{attribute 'GeneratedUsingTerminal: EP6002-0002-0023'}
{attribute addProperty BoxType "EP6002-0002-0023"}
{attribute addProperty Description "EP6002-0002 Interface (RS232/422/485)"}
{attribute addProperty Physics "YY"}
{attribute addProperty Id "COM_TxPDO_Map_Inputs_Channel_1AT %I*COM_TxPDO_Map_Inputs_Channel_6C2FC20224COM_TxPDO_Map_Inputs_Channel_2AT %I*COM_TxPDO_Map_Inputs_Channel_6C2FC20224COM_RxPDO_Map_Outputs_Channel_1AT %Q*COM_RxPDO_Map_Outputs_Channel_5D00B5E724COM_RxPDO_Map_Outputs_Channel_2AT %Q*COM_RxPDO_Map_Outputs_Channel_5D00B5E724WcStateAT %I*WcState_9091E0EB2InfoDataAT %I*InfoData_32EB74EA10"}
{attribute addProperty CRC "2078717463"}
{attribute addProperty Size "108"}
TYPE EP6002_7BE6B617 EXTENDS EtcSlaveBoxBase_77A0E4A7 :
STRUCT
	{attribute addProperty Name "COM_TxPDO_Map_Inputs_Channel_1"}
	COM_TxPDO_Map_Inputs_Channel_1 : COM_TxPDO_Map_Inputs_Channel_6C2FC202;
	{attribute addProperty Name "COM_TxPDO_Map_Inputs_Channel_2"}
	COM_TxPDO_Map_Inputs_Channel_2 : COM_TxPDO_Map_Inputs_Channel_6C2FC202;
	{attribute addProperty Name "COM_RxPDO_Map_Outputs_Channel_1"}
	COM_RxPDO_Map_Outputs_Channel_1 : COM_RxPDO_Map_Outputs_Channel_5D00B5E7;
	{attribute addProperty Name "COM_RxPDO_Map_Outputs_Channel_2"}
	COM_RxPDO_Map_Outputs_Channel_2 : COM_RxPDO_Map_Outputs_Channel_5D00B5E7;
	{attribute addProperty Name "WcState"}
	WcState : WcState_9091E0EB;
	{attribute addProperty Name "InfoData"}
	InfoData : InfoData_32EB74EA;
END_STRUCT
END_TYPE

(* stored: Version 1.2.0.0, ProductVersion 3.1.4024.11
   DUT EP6002_7BE6B617: Id {5698fd1b-6f29-4ca1-bdc8-8de6585df4db} *)
